{attribute 'qualified_only'}
VAR_GLOBAL CONSTANT
	MAX_NUMBER_OF_JOINTS : INT := 10; // 32 bit => max number is 2^32 - 1
END_VAR

(* stored: Version 1.1.0.1, ProductVersion 3.1.4024.9
   GVL GVL_RobotArmConstants: Id {7e4df322-2372-4313-a447-3a26c351e9c2} *)
